FUNCTION_BLOCK ADD_REMOVE_SLASH (* Basic Function Block Type *)
  (* Standard: 61499-2 *)
  (* Version 0.0, 20/01/2022, SESA489471, nxtControl GmbH, Template *)
  PACKAGE UAO.Hackathon;
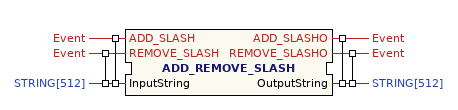
  EVENT_INPUT
    ADD_SLASH WITH InputString; (* Initialization Request *)
    REMOVE_SLASH WITH InputString; (* Normal Execution Request *)
  END_EVENT
  EVENT_OUTPUT
    ADD_SLASHO WITH OutputString; (* Initialization Confirm *)
    REMOVE_SLASHO WITH OutputString; (* Execution Confirmation *)
  END_EVENT
  VAR_INPUT
    InputString : STRING[512]; (* Input event qualifier *)
  END_VAR
  VAR_OUTPUT
    OutputString : STRING[512]; (* Output event qualifier *)
  END_VAR
  VAR
    Position : DINT;
    PositionTemp : DINT;
  END_VAR
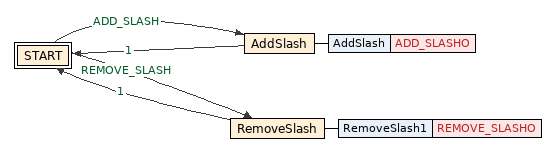
  EC_STATES
    START; (* Initial State *)
    AddSlash : AddSlash -> ADD_SLASHO; (* Initialization *)
    RemoveSlash : RemoveSlash1 -> REMOVE_SLASHO;
  END_STATES
  EC_TRANSITIONS
    START TO AddSlash := ADD_SLASH;
    AddSlash TO START := 1;
    START TO RemoveSlash := REMOVE_SLASH;
    RemoveSlash TO START := 1;
  END_TRANSITIONS
  ALGORITHM AddSlash IN ST: (* Initialization algorithm *)
OutputString := InputString;
Position := 0;
PositionTemp := 0;

PositionTemp:= FIND(InputString,'"');

WHILE PositionTemp <>0	DO
	Position := Position + PositionTemp - 1;
	OutputString := INSERT(OutputString,'\',Position);
	Position := Position +2; //slash is added

	InputString := DELETE(InputString,PositionTemp,1);
	PositionTemp:= FIND(InputString,'"');
END_WHILE;
  END_ALGORITHM
  ALGORITHM RemoveSlash1 IN ST: (* Normally executed algorithm *)
OutputString := InputString;
Position := 0;
PositionTemp := 0;

PositionTemp:= FIND(InputString,'\');

WHILE PositionTemp <>0	DO
	Position := Position + PositionTemp;

	OutputString := DELETE(OutputString,1,Position);
	Position := Position - 1; //slash is removed

	InputString := DELETE(InputString,PositionTemp,1);
	PositionTemp:= FIND(InputString,'\');
END_WHILE;

// for some reason Avahi function during the message parsing is adding additionally quotes (e.g.: "msg txt"),
 //which need to be removed, othervise JSON_PARSER can not decode the message

 OutputString := DELETE(OutputString,1,1);
 OutputString := DELETE(OutputString,1,LEN(OutputString));
  END_ALGORITHM
END_FUNCTION_BLOCK
